TYPE ST_Process_1_Measurements :
STRUCT
	//nID:			LINT;
	//tTime:		DATE_AND_TIME;
	sName:			STRING(50);
	fTemperature:	LREAL;
	fPressure:		LREAL;
	fFlowRate:		LREAL;
END_STRUCT
END_TYPE

(* stored: Version 1.1.0.1
   DUT ST_Process_1_Measurements: Id {7acde29a-c453-4510-8865-5b94d2d2fc86} *)
